// TIA Portal V17 export
// export: Created 2025-03-05T08:00:11.3053316Z, ExportSetting WithDefaults, DisplayName Totally Integrated Automation Portal, DisplayVersion V17 Update 8, DisplayName TIA Portal Openness, DisplayVersion V17 Update 8, DisplayName TIA Portal Version Control Interface, DisplayVersion V17, DisplayName SINAMICS Startdrive Advanced, DisplayVersion V17 SP2, DisplayName SINAMICS Startdrive G110M, G120, G120C, G120D, G120P, G115D, DisplayVersion V17 SP2, DisplayName SINAMICS Startdrive G130, G150, S120, S150, SINAMICS MV, S210, DisplayVersion V17 SP2, DisplayName STEP 7 Professional, DisplayVersion V17 Update 8, DisplayName SINUMERIK ONE STEP 7 Toolbox, DisplayVersion V17 Update 12, DisplayName SINUMERIK 840D sl STEP 7 Toolbox, DisplayVersion V17 Update 12, DisplayName STEP 7 Safety, DisplayVersion V17 Update 6, DisplayName WinCC Advanced, DisplayVersion V17 Update 8
FUNCTION "FC2101_LINE_CONTACTOR" : Void   // FC2101, LAD
{ S7_Optimized_Access := 'FALSE' }
AUTHOR : ETXETAR
VERSION : 1.0
// stored: AutoNumber false, IsIECCheckEnabled false, SetENOAutomatically false, UDAEnableTagReadback false
   VAR CONSTANT
      FC_NUMBER : DInt := 2101;   // FC NUMBER
   END_VAR
   VAR_TEMP   // added for the SCL form of the ladder/FBD networks
      _w1 : Bool;
      _w2 : Bool;
   END_VAR
BEGIN

REGION Network 1: OPTIONS OFF
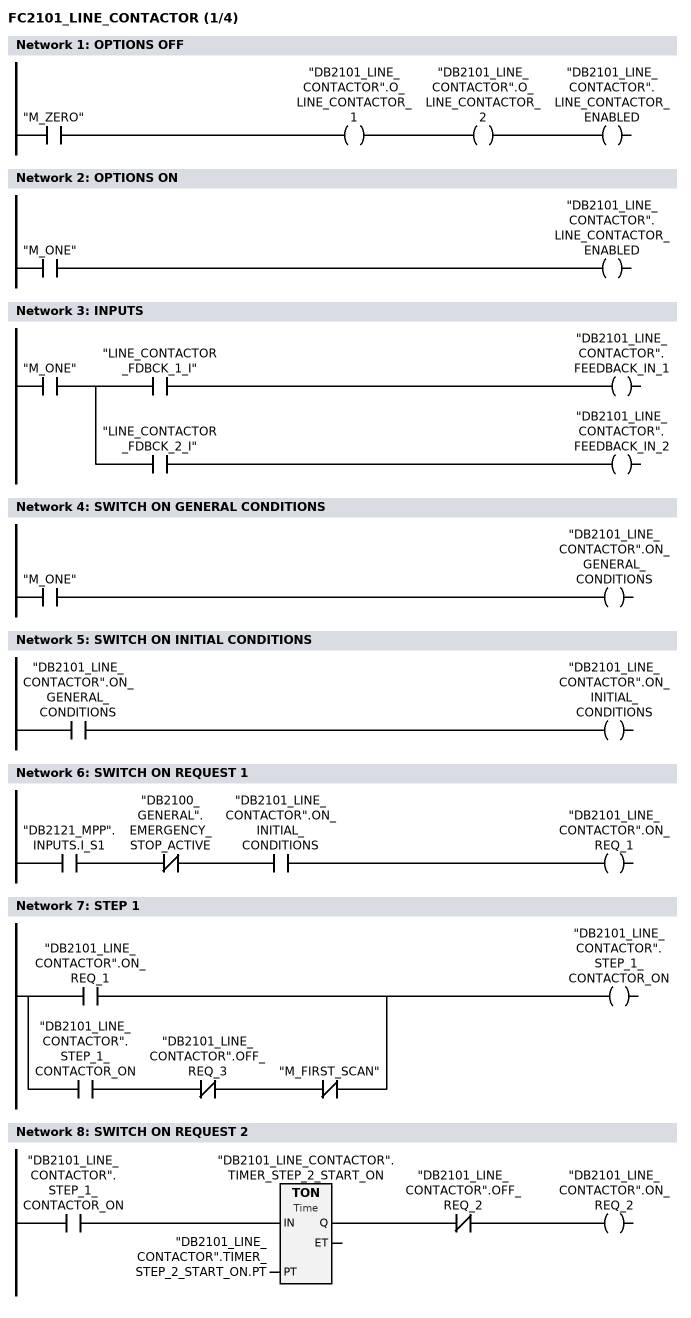
   RUNG wire#powerrail
      Contact( "M_ZERO" )
      Coil( "DB2101_LINE_CONTACTOR".O_LINE_CONTACTOR_1 )
      Coil( "DB2101_LINE_CONTACTOR".O_LINE_CONTACTOR_2 )
      Coil( "DB2101_LINE_CONTACTOR".LINE_CONTACTOR_ENABLED )
   END_RUNG
   // the same network as SCL:
   "DB2101_LINE_CONTACTOR".O_LINE_CONTACTOR_1 := "M_ZERO";
   "DB2101_LINE_CONTACTOR".O_LINE_CONTACTOR_2 := "M_ZERO";
   "DB2101_LINE_CONTACTOR".LINE_CONTACTOR_ENABLED := "M_ZERO";
END_REGION

REGION Network 2: OPTIONS ON
   RUNG wire#powerrail
      Contact( "M_ONE" )
      Coil( "DB2101_LINE_CONTACTOR".LINE_CONTACTOR_ENABLED )
   END_RUNG
   // the same network as SCL:
   "DB2101_LINE_CONTACTOR".LINE_CONTACTOR_ENABLED := "M_ONE";
END_REGION

REGION Network 3: INPUTS
   RUNG wire#powerrail
      Contact( "M_ONE" )
      wire#w1
      Contact( "LINE_CONTACTOR_FDBCK_1_I" )
      Coil( "DB2101_LINE_CONTACTOR".FEEDBACK_IN_1 )
   END_RUNG
   RUNG wire#w1
      Contact( "LINE_CONTACTOR_FDBCK_2_I" )
      Coil( "DB2101_LINE_CONTACTOR".FEEDBACK_IN_2 )
   END_RUNG
   // the same network as SCL:
   "DB2101_LINE_CONTACTOR".FEEDBACK_IN_1 := "M_ONE" AND "LINE_CONTACTOR_FDBCK_1_I";
   "DB2101_LINE_CONTACTOR".FEEDBACK_IN_2 := "M_ONE" AND "LINE_CONTACTOR_FDBCK_2_I";
END_REGION

REGION Network 4: SWITCH ON GENERAL CONDITIONS
   RUNG wire#powerrail
      Contact( "M_ONE" )
      Coil( "DB2101_LINE_CONTACTOR".ON_GENERAL_CONDITIONS )
   END_RUNG
   // the same network as SCL:
   "DB2101_LINE_CONTACTOR".ON_GENERAL_CONDITIONS := "M_ONE";
END_REGION

REGION Network 5: SWITCH ON INITIAL CONDITIONS
   RUNG wire#powerrail
      Contact( "DB2101_LINE_CONTACTOR".ON_GENERAL_CONDITIONS )
      Coil( "DB2101_LINE_CONTACTOR".ON_INITIAL_CONDITIONS )
   END_RUNG
   // the same network as SCL:
   "DB2101_LINE_CONTACTOR".ON_INITIAL_CONDITIONS := "DB2101_LINE_CONTACTOR".ON_GENERAL_CONDITIONS;
END_REGION

REGION Network 6: SWITCH ON REQUEST 1
   RUNG wire#powerrail
      Contact( "DB2121_MPP".INPUTS.I_S1 )
      I_Contact( "DB2100_GENERAL".EMERGENCY_STOP_ACTIVE )
      Contact( "DB2101_LINE_CONTACTOR".ON_INITIAL_CONDITIONS )
      Coil( "DB2101_LINE_CONTACTOR".ON_REQ_1 )
   END_RUNG
   // the same network as SCL:
   "DB2101_LINE_CONTACTOR".ON_REQ_1 := "DB2121_MPP".INPUTS.I_S1 AND NOT "DB2100_GENERAL".EMERGENCY_STOP_ACTIVE AND "DB2101_LINE_CONTACTOR".ON_INITIAL_CONDITIONS;
END_REGION

REGION Network 7: STEP 1
   RUNG wire#powerrail
      Contact( "DB2101_LINE_CONTACTOR".ON_REQ_1 )
      wire#w1
      Coil( "DB2101_LINE_CONTACTOR".STEP_1_CONTACTOR_ON )
   END_RUNG
   RUNG wire#powerrail
      Contact( "DB2101_LINE_CONTACTOR".STEP_1_CONTACTOR_ON )
      I_Contact( "DB2101_LINE_CONTACTOR".OFF_REQ_3 )
      I_Contact( "M_FIRST_SCAN" )
   END_RUNG wire#w1
   // the same network as SCL:
   "DB2101_LINE_CONTACTOR".STEP_1_CONTACTOR_ON := "DB2101_LINE_CONTACTOR".ON_REQ_1 OR ("DB2101_LINE_CONTACTOR".STEP_1_CONTACTOR_ON AND NOT "DB2101_LINE_CONTACTOR".OFF_REQ_3 AND NOT "M_FIRST_SCAN");
END_REGION

REGION Network 8: SWITCH ON REQUEST 2
   RUNG wire#powerrail
      Contact( "DB2101_LINE_CONTACTOR".STEP_1_CONTACTOR_ON )
      { S7_Templates := "time_type := Time" } "DB2101_LINE_CONTACTOR".TIMER_STEP_2_START_ON.TON(pt := "DB2101_LINE_CONTACTOR".TIMER_STEP_2_START_ON.PT, et =>)
      I_Contact( "DB2101_LINE_CONTACTOR".OFF_REQ_2 )
      Coil( "DB2101_LINE_CONTACTOR".ON_REQ_2 )
   END_RUNG
   // the same network as SCL:
   "DB2101_LINE_CONTACTOR".TIMER_STEP_2_START_ON.TON(IN := "DB2101_LINE_CONTACTOR".STEP_1_CONTACTOR_ON,
                           PT := "DB2101_LINE_CONTACTOR".TIMER_STEP_2_START_ON.PT);
   "DB2101_LINE_CONTACTOR".ON_REQ_2 := "DB2101_LINE_CONTACTOR".TIMER_STEP_2_START_ON.Q AND NOT "DB2101_LINE_CONTACTOR".OFF_REQ_2;
END_REGION

REGION Network 9: STEP 2
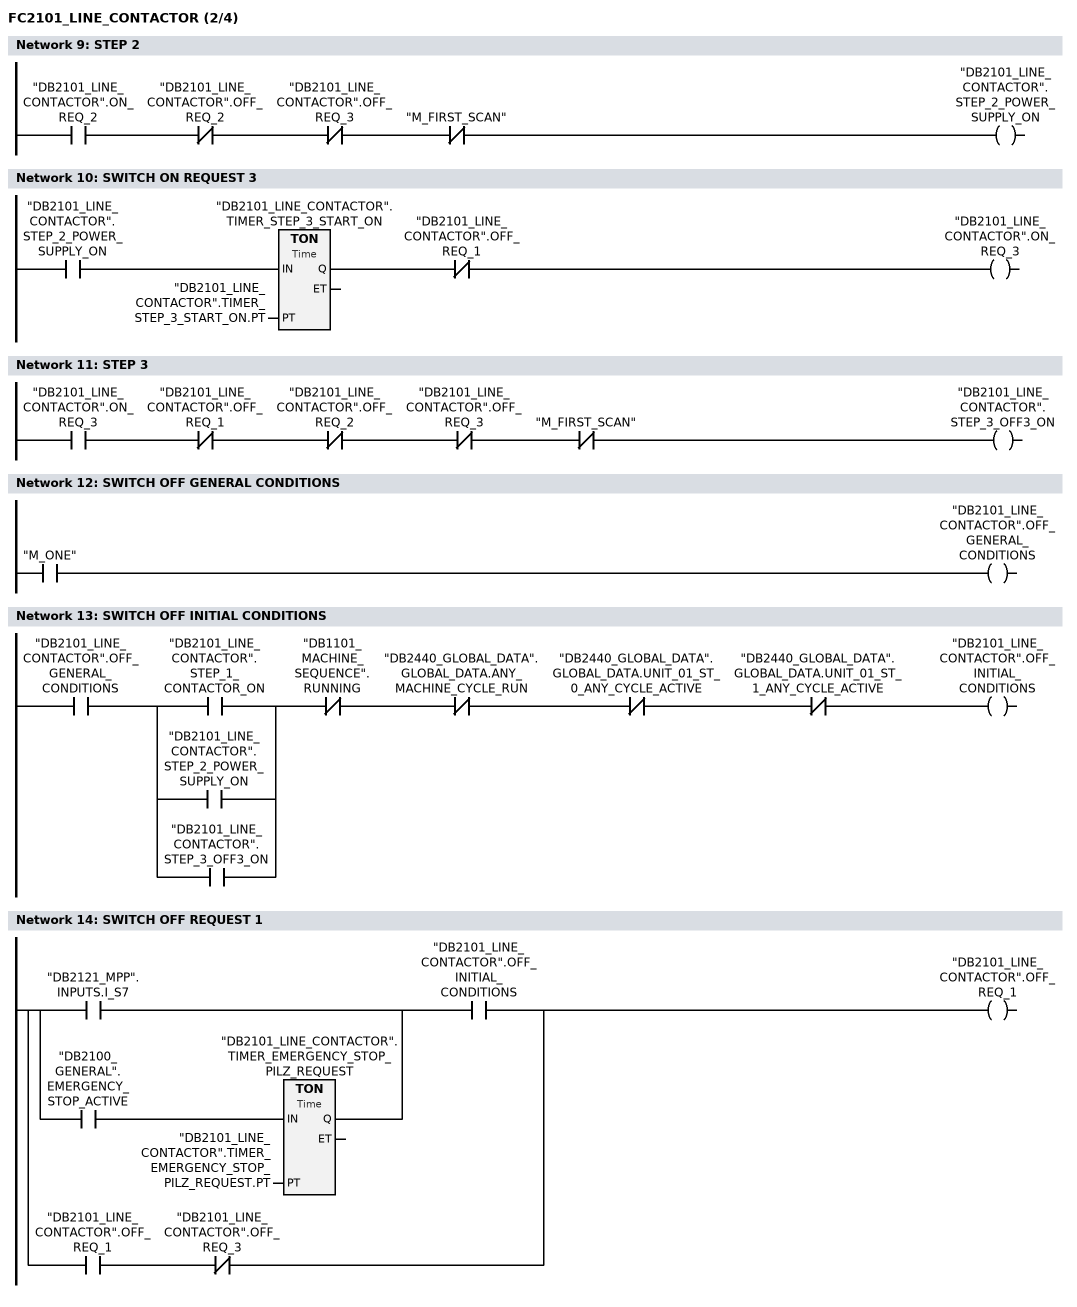
   RUNG wire#powerrail
      Contact( "DB2101_LINE_CONTACTOR".ON_REQ_2 )
      I_Contact( "DB2101_LINE_CONTACTOR".OFF_REQ_2 )
      I_Contact( "DB2101_LINE_CONTACTOR".OFF_REQ_3 )
      I_Contact( "M_FIRST_SCAN" )
      Coil( "DB2101_LINE_CONTACTOR".STEP_2_POWER_SUPPLY_ON )
   END_RUNG
   // the same network as SCL:
   "DB2101_LINE_CONTACTOR".STEP_2_POWER_SUPPLY_ON := "DB2101_LINE_CONTACTOR".ON_REQ_2 AND NOT "DB2101_LINE_CONTACTOR".OFF_REQ_2 AND NOT "DB2101_LINE_CONTACTOR".OFF_REQ_3 AND NOT "M_FIRST_SCAN";
END_REGION

REGION Network 10: SWITCH ON REQUEST 3
   RUNG wire#powerrail
      Contact( "DB2101_LINE_CONTACTOR".STEP_2_POWER_SUPPLY_ON )
      { S7_Templates := "time_type := Time" } "DB2101_LINE_CONTACTOR".TIMER_STEP_3_START_ON.TON(pt := "DB2101_LINE_CONTACTOR".TIMER_STEP_3_START_ON.PT, et =>)
      I_Contact( "DB2101_LINE_CONTACTOR".OFF_REQ_1 )
      Coil( "DB2101_LINE_CONTACTOR".ON_REQ_3 )
   END_RUNG
   // the same network as SCL:
   "DB2101_LINE_CONTACTOR".TIMER_STEP_3_START_ON.TON(IN := "DB2101_LINE_CONTACTOR".STEP_2_POWER_SUPPLY_ON,
                           PT := "DB2101_LINE_CONTACTOR".TIMER_STEP_3_START_ON.PT);
   "DB2101_LINE_CONTACTOR".ON_REQ_3 := "DB2101_LINE_CONTACTOR".TIMER_STEP_3_START_ON.Q AND NOT "DB2101_LINE_CONTACTOR".OFF_REQ_1;
END_REGION

REGION Network 11: STEP 3
   RUNG wire#powerrail
      Contact( "DB2101_LINE_CONTACTOR".ON_REQ_3 )
      I_Contact( "DB2101_LINE_CONTACTOR".OFF_REQ_1 )
      I_Contact( "DB2101_LINE_CONTACTOR".OFF_REQ_2 )
      I_Contact( "DB2101_LINE_CONTACTOR".OFF_REQ_3 )
      I_Contact( "M_FIRST_SCAN" )
      Coil( "DB2101_LINE_CONTACTOR".STEP_3_OFF3_ON )
   END_RUNG
   // the same network as SCL:
   "DB2101_LINE_CONTACTOR".STEP_3_OFF3_ON := "DB2101_LINE_CONTACTOR".ON_REQ_3 AND NOT "DB2101_LINE_CONTACTOR".OFF_REQ_1 AND NOT "DB2101_LINE_CONTACTOR".OFF_REQ_2 AND NOT "DB2101_LINE_CONTACTOR".OFF_REQ_3 AND NOT "M_FIRST_SCAN";
END_REGION

REGION Network 12: SWITCH OFF GENERAL CONDITIONS
   RUNG wire#powerrail
      Contact( "M_ONE" )
      Coil( "DB2101_LINE_CONTACTOR".OFF_GENERAL_CONDITIONS )
   END_RUNG
   // the same network as SCL:
   "DB2101_LINE_CONTACTOR".OFF_GENERAL_CONDITIONS := "M_ONE";
END_REGION

REGION Network 13: SWITCH OFF INITIAL CONDITIONS
   RUNG wire#powerrail
      Contact( "DB2101_LINE_CONTACTOR".OFF_GENERAL_CONDITIONS )
      wire#w1
      Contact( "DB2101_LINE_CONTACTOR".STEP_1_CONTACTOR_ON )
      wire#w2
      I_Contact( "DB1101_MACHINE_SEQUENCE".RUNNING )
      I_Contact( "DB2440_GLOBAL_DATA".GLOBAL_DATA.ANY_MACHINE_CYCLE_RUN )
      I_Contact( "DB2440_GLOBAL_DATA".GLOBAL_DATA.UNIT_01_ST_0_ANY_CYCLE_ACTIVE )
      I_Contact( "DB2440_GLOBAL_DATA".GLOBAL_DATA.UNIT_01_ST_1_ANY_CYCLE_ACTIVE )
      Coil( "DB2101_LINE_CONTACTOR".OFF_INITIAL_CONDITIONS )
   END_RUNG
   RUNG wire#w1
      Contact( "DB2101_LINE_CONTACTOR".STEP_2_POWER_SUPPLY_ON )
   END_RUNG wire#w2
   RUNG wire#w1
      Contact( "DB2101_LINE_CONTACTOR".STEP_3_OFF3_ON )
   END_RUNG wire#w2
   // the same network as SCL:
   "DB2101_LINE_CONTACTOR".OFF_INITIAL_CONDITIONS := "DB2101_LINE_CONTACTOR".OFF_GENERAL_CONDITIONS AND ("DB2101_LINE_CONTACTOR".STEP_1_CONTACTOR_ON OR "DB2101_LINE_CONTACTOR".STEP_2_POWER_SUPPLY_ON OR "DB2101_LINE_CONTACTOR".STEP_3_OFF3_ON) AND NOT "DB1101_MACHINE_SEQUENCE".RUNNING AND NOT "DB2440_GLOBAL_DATA".GLOBAL_DATA.ANY_MACHINE_CYCLE_RUN AND NOT "DB2440_GLOBAL_DATA".GLOBAL_DATA.UNIT_01_ST_0_ANY_CYCLE_ACTIVE AND NOT "DB2440_GLOBAL_DATA".GLOBAL_DATA.UNIT_01_ST_1_ANY_CYCLE_ACTIVE;
END_REGION

REGION Network 14: SWITCH OFF REQUEST 1
   RUNG wire#powerrail
      Contact( "DB2121_MPP".INPUTS.I_S7 )
      wire#w1
      Contact( "DB2101_LINE_CONTACTOR".OFF_INITIAL_CONDITIONS )
      wire#w2
      Coil( "DB2101_LINE_CONTACTOR".OFF_REQ_1 )
   END_RUNG
   RUNG wire#powerrail
      Contact( "DB2100_GENERAL".EMERGENCY_STOP_ACTIVE )
      { S7_Templates := "time_type := Time" } "DB2101_LINE_CONTACTOR".TIMER_EMERGENCY_STOP_PILZ_REQUEST.TON(pt := "DB2101_LINE_CONTACTOR".TIMER_EMERGENCY_STOP_PILZ_REQUEST.PT, et =>)
   END_RUNG wire#w1
   RUNG wire#powerrail
      Contact( "DB2101_LINE_CONTACTOR".OFF_REQ_1 )
      I_Contact( "DB2101_LINE_CONTACTOR".OFF_REQ_3 )
   END_RUNG wire#w2
   // the same network as SCL:
   "DB2101_LINE_CONTACTOR".TIMER_EMERGENCY_STOP_PILZ_REQUEST.TON(IN := "DB2100_GENERAL".EMERGENCY_STOP_ACTIVE,
                           PT := "DB2101_LINE_CONTACTOR".TIMER_EMERGENCY_STOP_PILZ_REQUEST.PT);
   "DB2101_LINE_CONTACTOR".OFF_REQ_1 := (("DB2121_MPP".INPUTS.I_S7 OR "DB2101_LINE_CONTACTOR".TIMER_EMERGENCY_STOP_PILZ_REQUEST.Q) AND "DB2101_LINE_CONTACTOR".OFF_INITIAL_CONDITIONS) OR ("DB2101_LINE_CONTACTOR".OFF_REQ_1 AND NOT "DB2101_LINE_CONTACTOR".OFF_REQ_3);
END_REGION

REGION Network 15: SWITCH OFF REQUEST 2
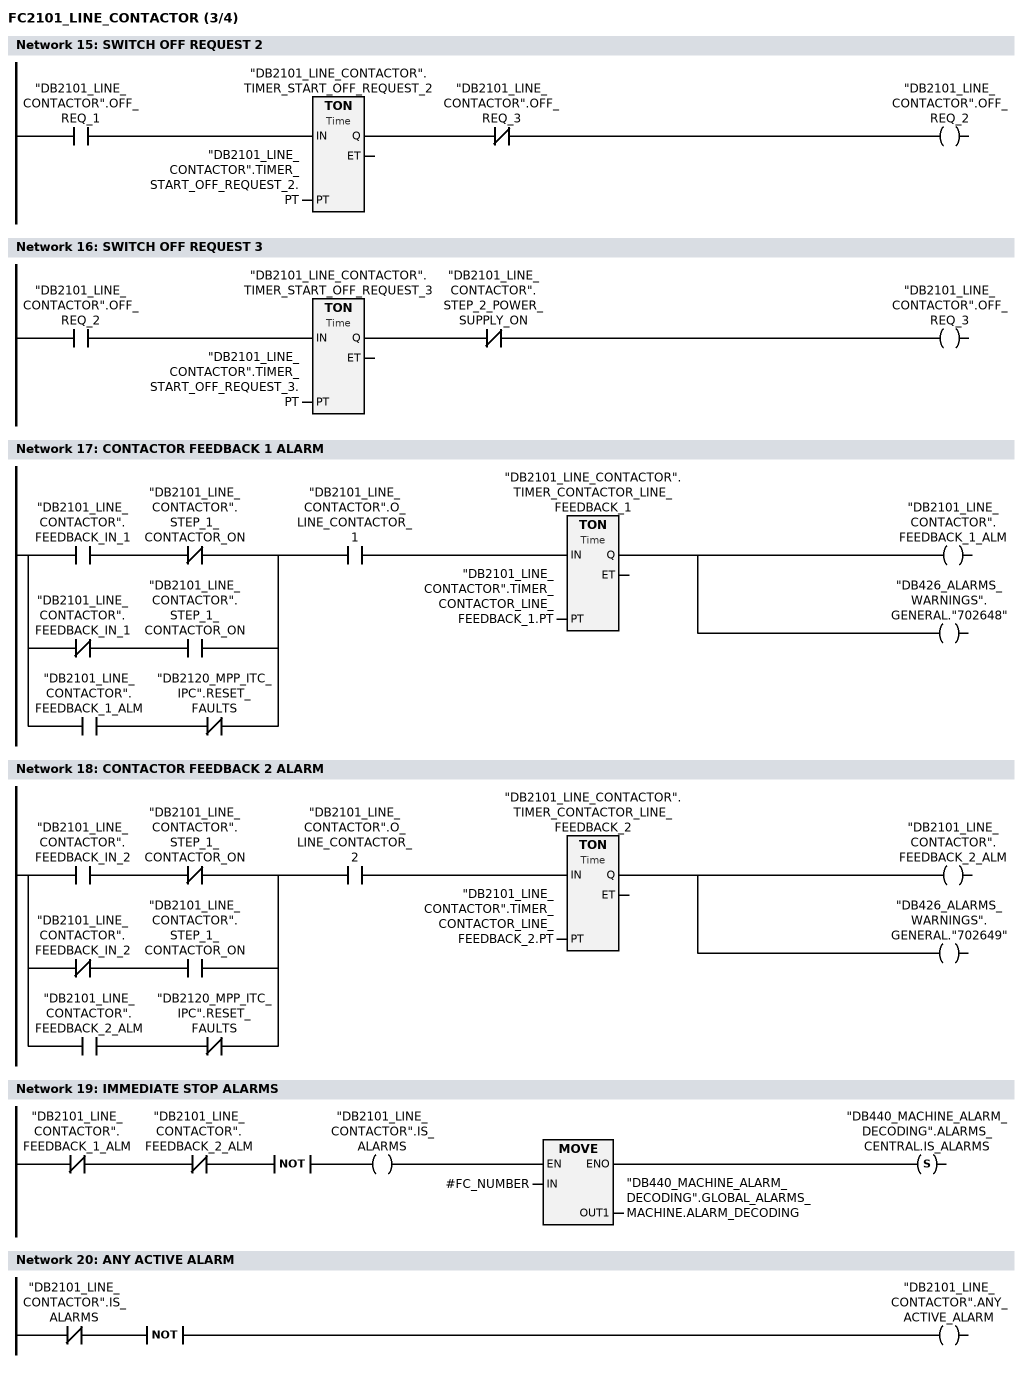
   RUNG wire#powerrail
      Contact( "DB2101_LINE_CONTACTOR".OFF_REQ_1 )
      { S7_Templates := "time_type := Time" } "DB2101_LINE_CONTACTOR".TIMER_START_OFF_REQUEST_2.TON(pt := "DB2101_LINE_CONTACTOR".TIMER_START_OFF_REQUEST_2.PT, et =>)
      I_Contact( "DB2101_LINE_CONTACTOR".OFF_REQ_3 )
      Coil( "DB2101_LINE_CONTACTOR".OFF_REQ_2 )
   END_RUNG
   // the same network as SCL:
   "DB2101_LINE_CONTACTOR".TIMER_START_OFF_REQUEST_2.TON(IN := "DB2101_LINE_CONTACTOR".OFF_REQ_1,
                           PT := "DB2101_LINE_CONTACTOR".TIMER_START_OFF_REQUEST_2.PT);
   "DB2101_LINE_CONTACTOR".OFF_REQ_2 := "DB2101_LINE_CONTACTOR".TIMER_START_OFF_REQUEST_2.Q AND NOT "DB2101_LINE_CONTACTOR".OFF_REQ_3;
END_REGION

REGION Network 16: SWITCH OFF REQUEST 3
   RUNG wire#powerrail
      Contact( "DB2101_LINE_CONTACTOR".OFF_REQ_2 )
      { S7_Templates := "time_type := Time" } "DB2101_LINE_CONTACTOR".TIMER_START_OFF_REQUEST_3.TON(pt := "DB2101_LINE_CONTACTOR".TIMER_START_OFF_REQUEST_3.PT, et =>)
      I_Contact( "DB2101_LINE_CONTACTOR".STEP_2_POWER_SUPPLY_ON )
      Coil( "DB2101_LINE_CONTACTOR".OFF_REQ_3 )
   END_RUNG
   // the same network as SCL:
   "DB2101_LINE_CONTACTOR".TIMER_START_OFF_REQUEST_3.TON(IN := "DB2101_LINE_CONTACTOR".OFF_REQ_2,
                           PT := "DB2101_LINE_CONTACTOR".TIMER_START_OFF_REQUEST_3.PT);
   "DB2101_LINE_CONTACTOR".OFF_REQ_3 := "DB2101_LINE_CONTACTOR".TIMER_START_OFF_REQUEST_3.Q AND NOT "DB2101_LINE_CONTACTOR".STEP_2_POWER_SUPPLY_ON;
END_REGION

REGION Network 17: CONTACTOR FEEDBACK 1 ALARM
   RUNG wire#powerrail
      Contact( "DB2101_LINE_CONTACTOR".FEEDBACK_IN_1 )
      I_Contact( "DB2101_LINE_CONTACTOR".STEP_1_CONTACTOR_ON )
      wire#w1
      Contact( "DB2101_LINE_CONTACTOR".O_LINE_CONTACTOR_1 )
      { S7_Templates := "time_type := Time" } "DB2101_LINE_CONTACTOR".TIMER_CONTACTOR_LINE_FEEDBACK_1.TON(pt := "DB2101_LINE_CONTACTOR".TIMER_CONTACTOR_LINE_FEEDBACK_1.PT, et =>)
      wire#w2
      Coil( "DB2101_LINE_CONTACTOR".FEEDBACK_1_ALM )
   END_RUNG
   RUNG wire#powerrail
      I_Contact( "DB2101_LINE_CONTACTOR".FEEDBACK_IN_1 )
      Contact( "DB2101_LINE_CONTACTOR".STEP_1_CONTACTOR_ON )
   END_RUNG wire#w1
   RUNG wire#powerrail
      Contact( "DB2101_LINE_CONTACTOR".FEEDBACK_1_ALM )
      I_Contact( "DB2120_MPP_ITC_IPC".RESET_FAULTS )
   END_RUNG wire#w1
   RUNG wire#w2
      Coil( "DB426_ALARMS_WARNINGS".GENERAL."702648" )
   END_RUNG
   // the same network as SCL:
   "DB2101_LINE_CONTACTOR".TIMER_CONTACTOR_LINE_FEEDBACK_1.TON(IN := (("DB2101_LINE_CONTACTOR".FEEDBACK_IN_1 AND NOT "DB2101_LINE_CONTACTOR".STEP_1_CONTACTOR_ON) OR (NOT "DB2101_LINE_CONTACTOR".FEEDBACK_IN_1 AND "DB2101_LINE_CONTACTOR".STEP_1_CONTACTOR_ON) OR ("DB2101_LINE_CONTACTOR".FEEDBACK_1_ALM AND NOT "DB2120_MPP_ITC_IPC".RESET_FAULTS)) AND "DB2101_LINE_CONTACTOR".O_LINE_CONTACTOR_1,
                           PT := "DB2101_LINE_CONTACTOR".TIMER_CONTACTOR_LINE_FEEDBACK_1.PT);
   "DB2101_LINE_CONTACTOR".FEEDBACK_1_ALM := "DB2101_LINE_CONTACTOR".TIMER_CONTACTOR_LINE_FEEDBACK_1.Q;
   "DB426_ALARMS_WARNINGS".GENERAL."702648" := "DB2101_LINE_CONTACTOR".TIMER_CONTACTOR_LINE_FEEDBACK_1.Q;
END_REGION

REGION Network 18: CONTACTOR FEEDBACK 2 ALARM
   RUNG wire#powerrail
      Contact( "DB2101_LINE_CONTACTOR".FEEDBACK_IN_2 )
      I_Contact( "DB2101_LINE_CONTACTOR".STEP_1_CONTACTOR_ON )
      wire#w1
      Contact( "DB2101_LINE_CONTACTOR".O_LINE_CONTACTOR_2 )
      { S7_Templates := "time_type := Time" } "DB2101_LINE_CONTACTOR".TIMER_CONTACTOR_LINE_FEEDBACK_2.TON(pt := "DB2101_LINE_CONTACTOR".TIMER_CONTACTOR_LINE_FEEDBACK_2.PT, et =>)
      wire#w2
      Coil( "DB2101_LINE_CONTACTOR".FEEDBACK_2_ALM )
   END_RUNG
   RUNG wire#powerrail
      I_Contact( "DB2101_LINE_CONTACTOR".FEEDBACK_IN_2 )
      Contact( "DB2101_LINE_CONTACTOR".STEP_1_CONTACTOR_ON )
   END_RUNG wire#w1
   RUNG wire#powerrail
      Contact( "DB2101_LINE_CONTACTOR".FEEDBACK_2_ALM )
      I_Contact( "DB2120_MPP_ITC_IPC".RESET_FAULTS )
   END_RUNG wire#w1
   RUNG wire#w2
      Coil( "DB426_ALARMS_WARNINGS".GENERAL."702649" )
   END_RUNG
   // the same network as SCL:
   "DB2101_LINE_CONTACTOR".TIMER_CONTACTOR_LINE_FEEDBACK_2.TON(IN := (("DB2101_LINE_CONTACTOR".FEEDBACK_IN_2 AND NOT "DB2101_LINE_CONTACTOR".STEP_1_CONTACTOR_ON) OR (NOT "DB2101_LINE_CONTACTOR".FEEDBACK_IN_2 AND "DB2101_LINE_CONTACTOR".STEP_1_CONTACTOR_ON) OR ("DB2101_LINE_CONTACTOR".FEEDBACK_2_ALM AND NOT "DB2120_MPP_ITC_IPC".RESET_FAULTS)) AND "DB2101_LINE_CONTACTOR".O_LINE_CONTACTOR_2,
                           PT := "DB2101_LINE_CONTACTOR".TIMER_CONTACTOR_LINE_FEEDBACK_2.PT);
   "DB2101_LINE_CONTACTOR".FEEDBACK_2_ALM := "DB2101_LINE_CONTACTOR".TIMER_CONTACTOR_LINE_FEEDBACK_2.Q;
   "DB426_ALARMS_WARNINGS".GENERAL."702649" := "DB2101_LINE_CONTACTOR".TIMER_CONTACTOR_LINE_FEEDBACK_2.Q;
END_REGION

REGION Network 19: IMMEDIATE STOP ALARMS
   RUNG wire#powerrail
      I_Contact( "DB2101_LINE_CONTACTOR".FEEDBACK_1_ALM )
      I_Contact( "DB2101_LINE_CONTACTOR".FEEDBACK_2_ALM )
      Not()
      Coil( "DB2101_LINE_CONTACTOR".IS_ALARMS )
      Move(in := #FC_NUMBER, out1 => "DB440_MACHINE_ALARM_DECODING".GLOBAL_ALARMS_MACHINE.ALARM_DECODING)
      S_Coil( "DB440_MACHINE_ALARM_DECODING".ALARMS_CENTRAL.IS_ALARMS )
   END_RUNG
   // the same network as SCL:
   "DB2101_LINE_CONTACTOR".IS_ALARMS := NOT (NOT "DB2101_LINE_CONTACTOR".FEEDBACK_1_ALM AND NOT "DB2101_LINE_CONTACTOR".FEEDBACK_2_ALM);
   IF "DB2101_LINE_CONTACTOR".IS_ALARMS THEN
       "DB440_MACHINE_ALARM_DECODING".GLOBAL_ALARMS_MACHINE.ALARM_DECODING := #FC_NUMBER;
       "DB440_MACHINE_ALARM_DECODING".ALARMS_CENTRAL.IS_ALARMS := TRUE;
   END_IF;
END_REGION

REGION Network 20: ANY ACTIVE ALARM
   RUNG wire#powerrail
      I_Contact( "DB2101_LINE_CONTACTOR".IS_ALARMS )
      Not()
      Coil( "DB2101_LINE_CONTACTOR".ANY_ACTIVE_ALARM )
   END_RUNG
   // the same network as SCL:
   "DB2101_LINE_CONTACTOR".ANY_ACTIVE_ALARM := NOT (NOT "DB2101_LINE_CONTACTOR".IS_ALARMS);
END_REGION

REGION Network 21: LINE CONTACTOR NOT SWITCHED ON WARNING
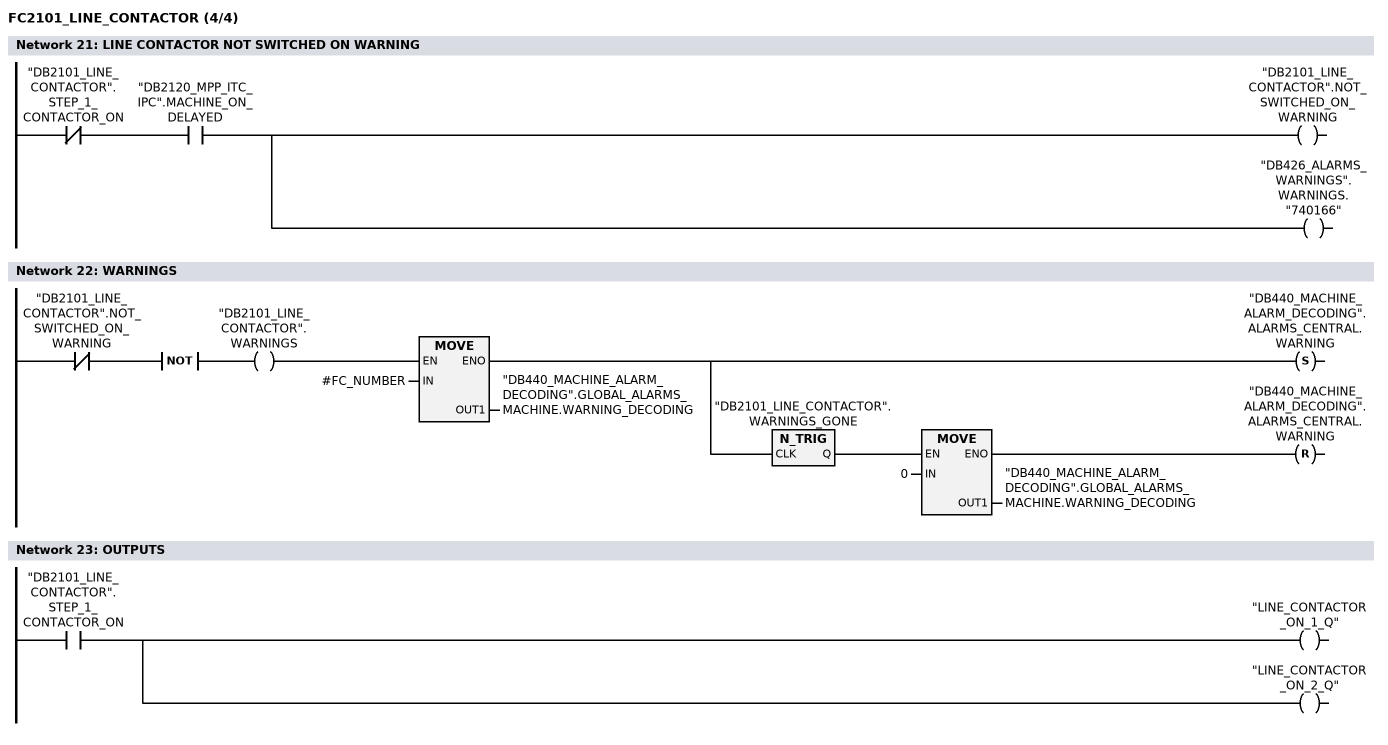
   RUNG wire#powerrail
      I_Contact( "DB2101_LINE_CONTACTOR".STEP_1_CONTACTOR_ON )
      Contact( "DB2120_MPP_ITC_IPC".MACHINE_ON_DELAYED )
      wire#w1
      Coil( "DB2101_LINE_CONTACTOR".NOT_SWITCHED_ON_WARNING )
   END_RUNG
   RUNG wire#w1
      Coil( "DB426_ALARMS_WARNINGS".WARNINGS."740166" )
   END_RUNG
   // the same network as SCL:
   "DB2101_LINE_CONTACTOR".NOT_SWITCHED_ON_WARNING := NOT "DB2101_LINE_CONTACTOR".STEP_1_CONTACTOR_ON AND "DB2120_MPP_ITC_IPC".MACHINE_ON_DELAYED;
   "DB426_ALARMS_WARNINGS".WARNINGS."740166" := "DB2101_LINE_CONTACTOR".NOT_SWITCHED_ON_WARNING;
END_REGION

REGION Network 22: WARNINGS
   RUNG wire#powerrail
      I_Contact( "DB2101_LINE_CONTACTOR".NOT_SWITCHED_ON_WARNING )
      Not()
      Coil( "DB2101_LINE_CONTACTOR".WARNINGS )
      Move(in := #FC_NUMBER, out1 => "DB440_MACHINE_ALARM_DECODING".GLOBAL_ALARMS_MACHINE.WARNING_DECODING)
      wire#w1
      S_Coil( "DB440_MACHINE_ALARM_DECODING".ALARMS_CENTRAL.WARNING )
   END_RUNG
   RUNG wire#w1
      N_Trig( "DB2101_LINE_CONTACTOR".WARNINGS_GONE )
      Move(in := 0, out1 => "DB440_MACHINE_ALARM_DECODING".GLOBAL_ALARMS_MACHINE.WARNING_DECODING)
      R_Coil( "DB440_MACHINE_ALARM_DECODING".ALARMS_CENTRAL.WARNING )
   END_RUNG
   // the same network as SCL:
   "DB2101_LINE_CONTACTOR".WARNINGS := NOT (NOT "DB2101_LINE_CONTACTOR".NOT_SWITCHED_ON_WARNING);
   #_w1 := NOT (NOT "DB2101_LINE_CONTACTOR".NOT_SWITCHED_ON_WARNING);
   IF #_w1 THEN
       "DB440_MACHINE_ALARM_DECODING".GLOBAL_ALARMS_MACHINE.WARNING_DECODING := #FC_NUMBER;
       "DB440_MACHINE_ALARM_DECODING".ALARMS_CENTRAL.WARNING := TRUE;
   END_IF;
   #_w2 := NOT #_w1 AND "DB2101_LINE_CONTACTOR".WARNINGS_GONE;   // falling edge
   "DB2101_LINE_CONTACTOR".WARNINGS_GONE := #_w1;
   IF #_w2 THEN
       "DB440_MACHINE_ALARM_DECODING".GLOBAL_ALARMS_MACHINE.WARNING_DECODING := 0;
       "DB440_MACHINE_ALARM_DECODING".ALARMS_CENTRAL.WARNING := FALSE;
   END_IF;
END_REGION

REGION Network 23: OUTPUTS
   RUNG wire#powerrail
      Contact( "DB2101_LINE_CONTACTOR".STEP_1_CONTACTOR_ON )
      wire#w1
      Coil( "LINE_CONTACTOR_ON_1_Q" )
   END_RUNG
   RUNG wire#w1
      Coil( "LINE_CONTACTOR_ON_2_Q" )
   END_RUNG
   // the same network as SCL:
   "LINE_CONTACTOR_ON_1_Q" := "DB2101_LINE_CONTACTOR".STEP_1_CONTACTOR_ON;
   "LINE_CONTACTOR_ON_2_Q" := "DB2101_LINE_CONTACTOR".STEP_1_CONTACTOR_ON;
END_REGION
END_FUNCTION
